# EPICS autosave request: support/calc-2-8/calcApp/Db/acalcoutArrays_settings.req
# FILE... acalcoutArrays_settings.req
# USAGE.. acalcout array fields autosave'd.

$(P).AA
$(P).BB
$(P).CC
$(P).DD
$(P).EE
$(P).FF
$(P).GG
$(P).HH
$(P).II
$(P).JJ
$(P).KK
$(P).LL
